{attribute addProperty BoxType "EL3204-0162-0016"}
{attribute addProperty Id "RTD_Inputs_ChannelAT %I*ARRAY[0..1] OF RTD_Inputs_Channel_F16A160D6480AI_Standard_ChannelAT %I*ARRAY[0..1] OF AI_Standard_Channel_5763EEB96480WcStateAT %I*WcState_F855686C1620InfoDataAT %I*InfoData_BC63D37F80100"}
{attribute addProperty CRC "578996451"}
{attribute addProperty SizeInBites "224"}
{attribute addProperty SizeInBytes "28"}
TYPE EL3204_34C8240A :
STRUCT
	{attribute addProperty Name "RTD_Inputs_Channel"}
	RTD_Inputs_Channel : ARRAY[0..1] OF RTD_Inputs_Channel_F16A160D;
	{attribute addProperty Name "AI_Standard_Channel"}
	AI_Standard_Channel : ARRAY[0..1] OF AI_Standard_Channel_5763EEB9;
	{attribute addProperty Name "WcState"}
	WcState : WcState_F855686C;
	{attribute addProperty Name "InfoData"}
	InfoData : InfoData_BC63D37F;
END_STRUCT
END_TYPE

(* stored: Version 1.2.0.0, ProductVersion 3.1.4024.9
   DUT EL3204_34C8240A: Id {50b3e496-a1df-48bd-80f9-243517645f26} *)
